FUNCTION_BLOCK ConveyorCTLMulti (* Basic Function Block Type *)
  (* Standard: 61499-2 *)
  (* Version 0.2, 2003-12-04, JHC, Rockwell Automation, Renamed for better indexing. *)
  (* Version 0.1, 2002-11-05, JHC, Rockwell Automation, Corrected missing ST element in Algorithm REQ. *)
  (* Version 0.0, 2000-05-30, JHC, Rockwell Automation *)
  (* Compiler header: package fb.rt.cs725; *)
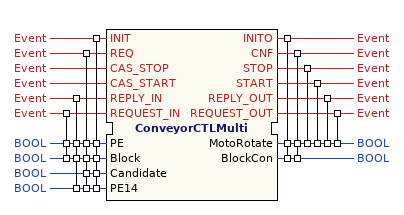
  EVENT_INPUT
    INIT WITH Block, Candidate, PE14, PE; (* Initialization Request *)
    REQ WITH PE, Block, Candidate, PE14; (* Normal Execution Request *)
    CAS_STOP;
    CAS_START;
    REPLY_IN WITH PE14, PE, Block;
    REQUEST_IN WITH PE, Block;
  END_EVENT
  EVENT_OUTPUT
    INITO WITH MotoRotate, BlockCon; (* Initialization Confirm *)
    CNF WITH MotoRotate, BlockCon; (* Execution Confirmation *)
    STOP WITH MotoRotate;
    START WITH MotoRotate;
    REPLY_OUT WITH MotoRotate;
    REQUEST_OUT WITH MotoRotate;
  END_EVENT
  VAR_INPUT
    PE : BOOL; (* Input event qualifier *)
    Block : BOOL;
    Candidate : BOOL;
    PE14 : BOOL;
  END_VAR
  VAR_OUTPUT
    MotoRotate : BOOL; (* Output event qualifier *)
    BlockCon : BOOL;
  END_VAR
  VAR
    lastPE : BOOL := 1;
    lastBlock : BOOL := 0;
    StoreEmit : BOOL := 0;
  END_VAR
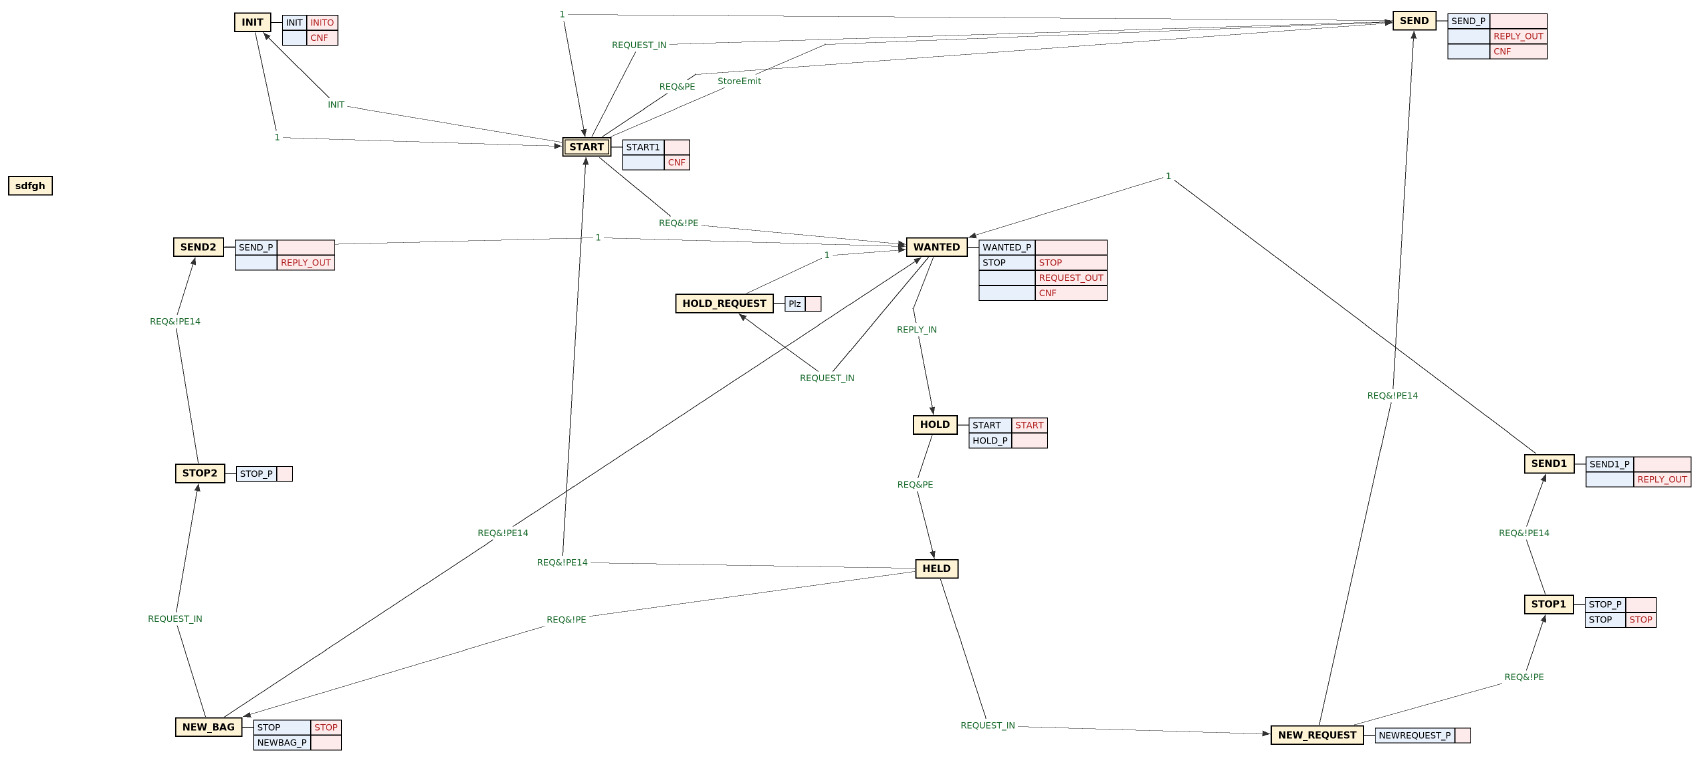
  EC_STATES
    START : START1, -> CNF; (* Initial State *)
    INIT : INIT -> INITO, -> CNF; (* Initialization *)
    SEND : SEND_P, -> REPLY_OUT, -> CNF;
    WANTED : WANTED_P, STOP -> STOP, -> REQUEST_OUT, -> CNF;
    NEW_BAG : STOP -> STOP, NEWBAG_P;
    NEW_REQUEST : NEWREQUEST_P;
    SEND2 : SEND_P, -> REPLY_OUT;
    STOP2 : STOP_P;
    HOLD : START -> START, HOLD_P;
    STOP1 : STOP_P, STOP -> STOP;
    SEND1 : SEND1_P, -> REPLY_OUT;
    HELD;
    HOLD_REQUEST : Plz;
    sdfgh;
  END_STATES
  EC_TRANSITIONS
    START TO INIT := INIT;
    INIT TO START := 1;
    START TO SEND := REQUEST_IN;
    SEND TO START := 1;
    START TO WANTED := REQ&!PE;
    NEW_REQUEST TO SEND := REQ&!PE14;
    STOP2 TO SEND2 := REQ&!PE14;
    SEND2 TO WANTED := 1;
    WANTED TO HOLD := REPLY_IN;
    STOP1 TO SEND1 := REQ&!PE14;
    SEND1 TO WANTED := 1;
    NEW_BAG TO STOP2 := REQUEST_IN;
    NEW_REQUEST TO STOP1 := REQ&!PE;
    HOLD TO HELD := REQ&PE;
    HELD TO NEW_BAG := REQ&!PE;
    HELD TO NEW_REQUEST := REQUEST_IN;
    HELD TO START := REQ&!PE14;
    NEW_BAG TO WANTED := REQ&!PE14;
    START TO SEND := REQ&PE;
    START TO SEND := StoreEmit;
    WANTED TO HOLD_REQUEST := REQUEST_IN;
    HOLD_REQUEST TO WANTED := 1;
  END_TRANSITIONS
  ALGORITHM INIT IN ST: (* Initialization algorithm *)
MotoRotate := TRUE;
Block := FALSE;

System.out.println(this + " " + MotoRotate);
System.out.println(MotoRotate);
  END_ALGORITHM
  ALGORITHM REQ IN ST: (* Normally executed algorithm *)
System.out.println(this +  " -> Candidate" + Candidate);
IF Candidate THEN
IF lastPE !:= PE THEN
IF NOT PE THEN
BlockCon:= TRUE;
System.out.println("BlockCon = true");
ELSE
BlockCon:=FALSE;
System.out.println("BlockCon = false");
END_IF
lastPE := PE;
END_IF
IF lastBlock !:= Block THEN
IF Block THEN
STOP.serviceEvent(this);
MotoRotate := FALSE;
System.out.println("Cas Stop");
ELSE
START.serviceEvent(this);
MotoRotate := TRUE;
System.out.println("Cas Start");
END_IF
lastBlock := Block;
END_IF
END_IF
  END_ALGORITHM
  ALGORITHM START IN ST:
MotoRotate:=TRUE;
System.out.println(this + " Start " + MotoRotate);

System.out.println("Start " + MotoRotate);

System.out.println("ENTERING CRITICAL SECTION");
  END_ALGORITHM
  ALGORITHM STOP IN ST:
MotoRotate := FALSE;
System.out.println(this + " Stop " + MotoRotate);

System.out.println("Stop " + MotoRotate);
System.out.println("IN WAITING");
  END_ALGORITHM
  ALGORITHM print IN ST:
System.out.println(this + "IM here");
  END_ALGORITHM
  ALGORITHM START1 IN Java:
System.out.println("START STATE");
  END_ALGORITHM
  ALGORITHM SEND_P IN Java:
System.out.println("SEND STATE");
  END_ALGORITHM
  ALGORITHM WANTED_P IN Java:
System.out.println("WANTED STATE");
  END_ALGORITHM
  ALGORITHM HELD_P IN Java:
System.out.println("HELD STATE");
  END_ALGORITHM
  ALGORITHM NEWBAG_P IN Java:
System.out.println("NEWBAG STATE");
  END_ALGORITHM
  ALGORITHM NEWREQUEST_P IN Java:
System.out.println("NEWREQUEST STATE");
  END_ALGORITHM
  ALGORITHM SEND1_P IN Java:
System.out.println("SEND1 STATE");
  END_ALGORITHM
  ALGORITHM STOP_P IN Java:
System.out.println("STOP STATE");
  END_ALGORITHM
  ALGORITHM HOLD_P IN Java:
System.out.println("HOLD STATE");
  END_ALGORITHM
  ALGORITHM NEW_REQUEST2_P IN Java:
System.out.println("NEW_REQUEST2 STATE");
  END_ALGORITHM
  ALGORITHM Plz IN ST:
StoreEmit := TRUE;
  END_ALGORITHM
  ALGORITHM not_plz IN ST:
StoreEmit := FALSE;
  END_ALGORITHM
END_FUNCTION_BLOCK
